PROGRAM MAIN
VAR
	CounterFromUser1	: DINT;
END_VAR

CounterFromUser1	:= CounterFromUser1 +2;

END_PROGRAM

(* stored: Version 1.1.0.1, ProductVersion 3.1.4026.13
   POU MAIN: Id {185222de-2f69-4bea-a76f-3614533a9172}, SpecialFunc None *)
